FUNCTION_BLOCK ShutterSwitch

VAR CONSTANT
	MAX_OUTPUTS_PER_LEVEL : INT := 2;
END_VAR

VAR_INPUT
	ID : INT;
	name : STRING := "Shutter switch";
	digitalInputUp : REFERENCE TO BOOL;
	digitalInputDown : REFERENCE TO BOOL;
	up_outputs : REFERENCE TO ARRAY[1..MAX_OUTPUTS_PER_LEVEL] OF BOOL;
	down_outputs : REFERENCE TO ARRAY[1..MAX_OUTPUTS_PER_LEVEL] OF BOOL;
END_VAR

VAR_OUTPUT
END_VAR

VAR
	isClosing : BOOL := FALSE;
	isOpening : BOOL := FALSE;
	
    pressedUp : R_TRIG;
	pressedDown : R_TRIG;
	releasedUp : F_TRIG;
	releasedDown : F_TRIG;
	
	pressedUpTimer : TON := (PT := T#10S);	
	pressedDownTimer : TON := (PT := T#10S);
	
	shortDistanceUp : TP := (PT := T#200MS);
	longDistanceUp : TP := (PT := T#60S);
	shortDistanceDown : TP := (PT := T#200MS);
	longDistanceDown : TP := (PT := T#60S);
	
	initialized : BOOL := FALSE;
	
	pressedUpMiliseconds : INT := 0;
	pressedDownMiliseconds : INT := 0;	
	
	goUpRequested : BOOL := FALSE;
	goDownRequested : BOOL := FALSE;
	
	canPrintGoUp : BOOL := TRUE;
	canPrintGoDown : BOOL := TRUE;
END_VAR

IF NOT initialized THEN
	initialized := TRUE;	
END_IF

METHOD getSource : STRING
VAR_INPUT
END_VAR

VAR
	details : STRING;
END_VAR
details := CONCAT(STR1:=' - shutter switch, ID: ', STR2:=TO_STRING(ID));
details := CONCAT(STR1:=details, STR2:=', digital input up: ');
details := CONCAT(STR1:=details, STR2:=TO_STRING(digitalInputUp));
details := CONCAT(STR1:=details, STR2:=', digital input down: ');
details := CONCAT(STR1:=details, STR2:=TO_STRING(digitalInputDown));
details := CONCAT(STR1:=details, STR2:=', name: ');
details := CONCAT(STR1:=details, STR2:=name);
END_METHOD

METHOD loop : BOOL
VAR_INPUT
END_VAR

VAR
END_VAR
pressedUp(CLK:= digitalInputUp);
pressedDown(CLK:= digitalInputDown);
releasedUp(CLK:= digitalInputUp);
releasedDown(CLK:= digitalInputDown);
pressedUpTimer(IN := digitalInputUp);
pressedDownTimer(IN := digitalInputDown);

//prevent both pressed
IF digitalInputUp AND digitalInputDown THEN
	GVL.EventLogger.print3(level:=TcEventSeverity.Warning, str1:='Both button pressed', str2:='', str3:=getSource);
	stopAll();
	pressedUpMiliseconds := 0;
	pressedDownMiliseconds := 0;
	JMP _ret;
END_IF

//moving any direction 
IF isClosing OR isOpening THEN
	IF pressedUp.Q OR pressedDown.Q THEN
		GVL.EventLogger.print3(level:=TcEventSeverity.Info, str1:='Button pressed during shutter move', str2:='', str3:=getSource);
		stopAll();
		JMP _ret;
	END_IF
END_IF

goUpRequested := shortDistanceUp.Q OR longDistanceUp.Q;
goDownRequested := shortDistanceDown.Q OR longDistanceDown.Q;
IF goUpRequested AND NOT goDownRequested THEN
	moveUp();
ELSE 
	stopUp();
END_IF

IF goDownRequested AND NOT goUpRequested THEN
	moveDown();
ELSE 
	stopDown();
END_IF

//long hold up
IF digitalInputUp AND TIME_TO_INT(pressedUpTimer.ET) <> 0 THEN
	pressedUpMiliseconds := TIME_TO_INT(pressedUpTimer.ET);
END_IF

//long hold downm
IF digitalInputDown AND TIME_TO_INT(pressedDownTimer.ET) <> 0 THEN
	pressedDownMiliseconds := TIME_TO_INT(pressedDownTimer.ET);
END_IF

IF releasedUp THEN
	GVL.EventLogger.print3(level:=TcEventSeverity.Verbose, str1:='Button up released after ', str2:=TO_STRING(pressedUpMiliseconds), str3:=getSource);
	onReleasedUp();
END_IF

IF pressedUpMiliseconds >= 2000 THEN
	moveUp();
END_IF

IF releasedDown THEN
	GVL.EventLogger.print3(level:=TcEventSeverity.Verbose, str1:='Button down released after ', str2:=TO_STRING(pressedDownMiliseconds), str3:=getSource);
	onReleasedDown();
END_IF

IF pressedDownMiliseconds >= 2000 THEN
	moveDown();
END_IF

_ret :
END_METHOD

METHOD moveDown : BOOL
VAR_INPUT
END_VAR
IF canPrintGoDown THEN
	GVL.EventLogger.print3(level:=TcEventSeverity.Info, str1:='Roller shutter moving down', str2:='', str3:=getSource);
	canPrintGoDown := FALSE;
END_IF
setOutputs(direction:=E_Direction.UP, state:=FALSE);
setOutputs(direction:=E_Direction.DOWN, state:=TRUE);
END_METHOD

METHOD moveUp : BOOL
VAR_INPUT
END_VAR
IF canPrintGoUp THEN
	GVL.EventLogger.print3(level:=TcEventSeverity.Info, str1:='Roller shutter moving up', str2:='', str3:=getSource);
	canPrintGoUp := FALSE;
END_IF

setOutputs(direction:=E_Direction.DOWN, state:=FALSE);
setOutputs(direction:=E_Direction.UP, state:=TRUE);
END_METHOD

METHOD onReleasedDown : BOOL
VAR_INPUT
END_VAR
GVL.EventLogger.print3(level:=TcEventSeverity.Verbose, str1:='pressedDownMiliseconds=', str2:= TO_STRING(pressedDownMiliseconds), str3:=getSource);

IF pressedDownMiliseconds > 10 AND pressedDownMiliseconds < 500 THEN
	//move a bit down
	shortDistanceDown(IN:=TRUE);
ELSIF pressedDownMiliseconds >= 500 AND pressedDownMiliseconds < 2000 THEN
	//move max down
	longDistanceDown(IN:=TRUE);
ELSIF pressedDownMiliseconds >= 2000 THEN
	//stop
	stopAll();
END_IF

pressedDownMiliseconds := 0;
END_METHOD

METHOD onReleasedUp : BOOL
VAR_INPUT
END_VAR
GVL.EventLogger.print3(level:=TcEventSeverity.Verbose, str1:='pressedUpMiliseconds=', str2:= TO_STRING(pressedUpMiliseconds), str3:=getSource);

IF pressedUpMiliseconds > 10 AND pressedUpMiliseconds < 500 THEN
	//move a little bit up
	shortDistanceUp(IN:=TRUE);
ELSIF pressedUpMiliseconds >= 500 AND pressedUpMiliseconds < 2000 THEN
	//move max up
	longDistanceUp(IN:=TRUE);
ELSIF pressedUpMiliseconds >= 2000 THEN
	//stop
	stopAll();
END_IF

pressedUpMiliseconds := 0;
END_METHOD

METHOD setOutputs
VAR_INPUT
	direction : E_Direction;
	state : BOOL;
END_VAR

VAR
	i : INT;
	state_as_text : STRING := 'abc';
END_VAR
state_as_text := TO_STRING(state);

CASE direction OF
	
	E_Direction.UP:
		GVL.EventLogger.print3(level:=TcEventSeverity.Info, str1:='set UP to: ', str2:= state_as_text, str3:=getSource);
		FOR i := 1 TO MAX_OUTPUTS_PER_LEVEL BY 1 DO
			up_outputs[i] := state;
		END_FOR
		
	E_Direction.DOWN:
		GVL.EventLogger.print3(level:=TcEventSeverity.Info, str1:='set DOWN to: ', str2:= state_as_text, str3:=getSource);	
		FOR i := 1 TO MAX_OUTPUTS_PER_LEVEL BY 1 DO
			down_outputs[i] := state;
		END_FOR
		
END_CASE
END_METHOD

METHOD stopAll : BOOL
VAR_INPUT
END_VAR
GVL.EventLogger.print3(level:=TcEventSeverity.Info, str1:='Stopping roller shutter', str2:='', str3:=getSource);
stopDown();
stopUp();
END_METHOD

METHOD stopDown : BOOL
VAR_INPUT
END_VAR
GVL.EventLogger.print3(level:=TcEventSeverity.Info, str1:='Roller shutter moving down stopped', str2:='', str3:=getSource);
canPrintGoDown := TRUE;
setOutputs(direction:=E_Direction.DOWN, state:=FALSE);
END_METHOD

METHOD stopUp : BOOL
VAR_INPUT
END_VAR
GVL.EventLogger.print3(level:=TcEventSeverity.Info, str1:='Roller shutter moving up stopped', str2:='', str3:=getSource);
canPrintGoUp := TRUE;
setOutputs(direction:=E_Direction.UP, state:=FALSE);
END_METHOD

END_FUNCTION_BLOCK

(* stored: Version 1.1.0.1, ProductVersion 3.1.4024.12
   POU ShutterSwitch: Id {ea3d4221-9f14-4b85-9e8e-0f11bb1f6816}, SpecialFunc None
   Method getSource: Id {3343044d-517d-47e0-899f-f77bf241ae33}
   Method loop: Id {9386c37e-49fd-4cf9-895c-78c751a8bca5}
   Method moveDown: Id {70bfc2f0-2a45-495c-8a8c-08f2039c444b}
   Method moveUp: Id {be6ff087-74af-4f3e-8a6d-a69e0bda1f40}
   Method onReleasedDown: Id {d189a28a-8b68-42c4-b7ce-29fd95d074d7}
   Method onReleasedUp: Id {18137760-a3db-4047-aa6a-2ed70d4a3ef6}
   Method setOutputs: Id {79b15e5b-fc69-4f91-8345-898161fcd2f3}
   Method stopAll: Id {69f3a6d7-377a-4aed-9325-e1404881787f}
   Method stopDown: Id {e9b25731-7d10-4d84-bd86-0f94bf8f47e3}
   Method stopUp: Id {d5b93eb4-00aa-4364-a9b2-6f05420d9e05} *)
